TYPE ST_RFID_DATA :
STRUCT
	aRFIDData:		ARRAY[1..8] OF USINT;
	nPalletID:		UDINT;
	sRecipeName:	STRING;
END_STRUCT
END_TYPE

(* stored: Version 1.1.0.1, ProductVersion 3.1.4024.12
   DUT ST_RFID_DATA: Id {d415cb34-051c-4c66-8835-fd3aa844ade8} *)
